PROGRAM Auto_Mode
VAR_INPUT
	SFCPause:BOOL;
	SFCCurrentStep:STRING;
	SFCInit:BOOL;
END_VAR
VAR
	Activator: INT;
END_VAR

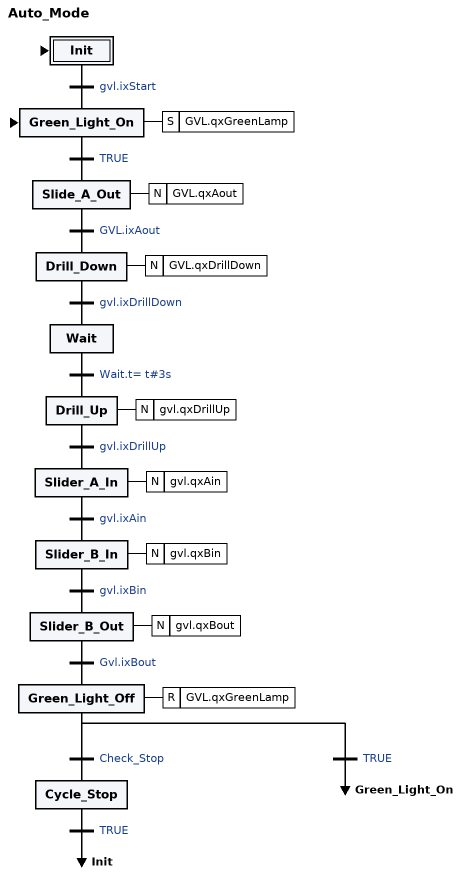
INITIAL_STEP Init:
END_STEP
TRANSITION FROM Init TO Green_Light_On
    := gvl.ixStart;
END_TRANSITION
STEP Green_Light_On:
    GVL.qxGreenLamp(S);
END_STEP
TRANSITION FROM Green_Light_On TO Slide_A_Out
    := TRUE;
END_TRANSITION
STEP Slide_A_Out:
    GVL.qxAout(N);
END_STEP
TRANSITION FROM Slide_A_Out TO Drill_Down
    := GVL.ixAout;
END_TRANSITION
STEP Drill_Down:
    GVL.qxDrillDown(N);
END_STEP
TRANSITION FROM Drill_Down TO Wait
    := gvl.ixDrillDown;
END_TRANSITION
STEP Wait:
END_STEP
TRANSITION FROM Wait TO Drill_Up
    := Wait.t= t#3s;
END_TRANSITION
STEP Drill_Up:
    gvl.qxDrillUp(N);
END_STEP
TRANSITION FROM Drill_Up TO Slider_A_In
    := gvl.ixDrillUp;
END_TRANSITION
STEP Slider_A_In:
    gvl.qxAin(N);
END_STEP
TRANSITION FROM Slider_A_In TO Slider_B_In
    := gvl.ixAin;
END_TRANSITION
STEP Slider_B_In:
    gvl.qxBin(N);
END_STEP
TRANSITION FROM Slider_B_In TO Slider_B_Out
    := gvl.ixBin;
END_TRANSITION
STEP Slider_B_Out:
    gvl.qxBout(N);
END_STEP
TRANSITION FROM Slider_B_Out TO Green_Light_Off
    := Gvl.ixBout;
END_TRANSITION
STEP Green_Light_Off:
    GVL.qxGreenLamp(R);
END_STEP
TRANSITION FROM Green_Light_Off TO Cycle_Stop
    := Check_Stop;
END_TRANSITION
STEP Cycle_Stop:
END_STEP
TRANSITION FROM Cycle_Stop TO Init
    := TRUE;
END_TRANSITION
TRANSITION FROM Green_Light_Off TO Green_Light_On
    := TRUE;
END_TRANSITION

TRANSITION Check_Stop:
IF gvl.ixStop THEN
	Activator:= 1;
END_IF
IF Activator=1 THEN
	Check_Stop:=TRUE;
END_IF
IF gvl.ixStart THEN
	Activator:= 0;
	Check_Stop:=FALSE;
END_IF
END_TRANSITION

END_PROGRAM

(* stored: Version 1.1.0.1, ProductVersion 3.1.4024.12
   POU Auto_Mode: Id {45f1c680-b9ee-438c-a695-08fcadf0b1c0}, SpecialFunc None
   Transition Check_Stop: Id {31ae41c4-d674-4b00-94eb-68d35e576bdc} *)
